// SIMATIC S7-200 project (STEP 7-Micro/WIN), CPU 224 REL 02.01

ORGANIZATION_BLOCK MAIN:OB1
TITLE=PROGRAM COMMENTS
BEGIN
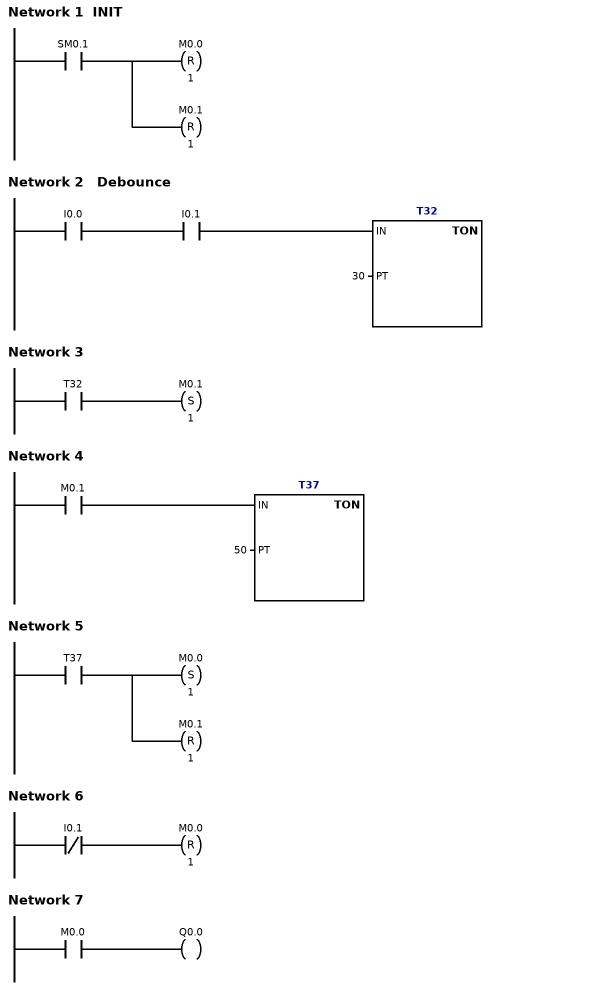
Network 1 // INIT
// (network saved uncompiled; LAD cells follow)
// row 0: c0 -| |- SM0.1 v  c1 -(R) M0.0, 1
// row 1: c0 ^  c1 -(R) M0.1, 1
Network 2 //  Debounce 
LD     I0.0
A      I0.1
TON    T32, 30
Network 3
LD     T32
S      M0.1, 1
Network 4
LD     M0.1
TON    T37, 50
Network 5
LD     T37
S      M0.0, 1
R      M0.1, 1
Network 6
LDN    I0.1
R      M0.0, 1
Network 7
LD     M0.0
=      Q0.0
END_ORGANIZATION_BLOCK
